// TIA Portal V18 export
DATA_BLOCK "TCSData"   // DB4
{ S7_Optimized_Access := 'TRUE' }
VERSION : 0.1
// stored: AutoNumber true, DBAccessibleFromOPCUA true, IsOnlyStoredInLoadMemory false, IsRetainMemResEnabled false, IsWriteProtectedInAS false, MemoryReserve 100
   VAR
      Data : Array[0..1] of Word;
      Connect : TCON_IP_v4;
   END_VAR
BEGIN
   Connect.InterfaceId := 64;
   Connect.ID := 16#1;
   Connect.LocalPort := 502;
END_DATA_BLOCK
